{attribute 'Tc2GvlVarNames'}
{attribute 'strict'}
//Stato del WorkAreaManager
TYPE e_Stato_WorkArea :
(
	WORKAREA_STATE_FREE_ENABLED					:= 0,	//WA senza pallet e Abilitata
	WORKAREA_STATE_FREE_DISABLED				:= 1,	//WA senza pallet e disabilitata
	WORKAREA_STATE_OCCUPIED_DISABLED			:= 2,	//WA con pallet e disabilitata
	WORKAREA_STATE_FREE_WORKING					:= 3,	//WA senza pallet e in lavorazione
	WORKAREA_STATE_OCCUPIED_WORKING				:= 4,	//WA con pallet e in lavorazione	
	WORKAREA_STATE_OCCUPIED_WORKED				:= 5, 	//WA con pallet e pallettizzazione terminata
	WORKAREA_STATE_OCCUPIED_WORKED_DISABLED		:= 6,	//WA con pallet e pallettizzazione terminata e area disabilitata
	WORKAREA_STATE_OCCUPIED_TAPING				:= 7,	//WA con pallet in richiesta di nastratura
	WORKAREA_STATE_OCCUPIED_TAPING_DISABLED		:= 8,	//WA con pallet in richiesta di nastratura e area disabilitata
	WORKAREA_STATE_OCCUPIED_TAPED				:= 9,	//WA con pallet e nastratura terminata
	WORKAREA_STATE_OCCUPIED_TAPED_DISABLED		:= 10,	//WA con pallet e nastratura terminata e area disabilitata
	WORKAREA_STATE_OCCUPIED_ENDED				:= 11, 	//WA con pallet e lavorazione terminata
	WORKAREA_STATE_OCCUPIED_ENDED_DISABLED		:= 12, 	//WA con pallet e lavorazione terminata e area disabilitata
	WORKAREA_STATE_OCCUPIED_LGVREQ				:= 13, 	//WA con pallet e richiesta TGV in ingresso
	WORKAREA_STATE_OCCUPIED_LGVREQ_DISABLED		:= 14, 	//WA con pallet e richiesta TGV in ingresso e area disabilitata
	WORKAREA_STATE_OCCUPIED_LGVIN				:= 15, 	//WA con pallet e TGV in ingombro
	WORKAREA_STATE_OCCUPIED_LGVIN_DISABLED		:= 16, 	//WA con pallet e TGV in ingombro e area disabilitata
	WORKAREA_STATE_OCCUPIED_LGVEND				:= 17, 	//WA con pallet e TGV fuori ingombro e Pallet estratto
	WORKAREA_STATE_OCCUPIED_LGVEND_DISABLED		:= 18, 	//WA con pallet e TGV fuori ingombro e Pallet estratto e area disabilata
	WORKAREA_STATE_OCCUPIED_LGVREQ_ABORT        := 19, 	//WA con pallet e richiesta TGV ABORTITA
	
	WORKAREA_STATE_FREE_LGVREQ					:= 20, 	//WA SENZA SUPPORTO e richiesta TGV in ingresso
	WORKAREA_STATE_FREE_LGVREQ_DISABLED			:= 21, 	//WA SENZA SUPPORTO e richiesta TGV in ingresso e area disabilitata
	WORKAREA_STATE_FREE_LGVIN					:= 22, 	//WA SENZA SUPPORTO e TGV in ingombro
	WORKAREA_STATE_FREE_LGVIN_DISABLED			:= 23, 	//WA SENZA SUPPORTO e TGV in ingombro e area disabilitata
	WORKAREA_STATE_FREE_LGVEND					:= 24, 	//WA SENZA SUPPORTO e TGV fuori ingombro e Pallet estratto
	WORKAREA_STATE_FREE_LGVEND_DISABLED			:= 25, 	//WA SENZA SUPPORTO e TGV fuori ingombro e Pallet estratto e area disabilata
	WORKAREA_STATE_FREE_LGVREQ_ABORT        	:= 26, 	//WA SENZA SUPPORTO e richiesta TGV ABORTITA
	
	WORKAREA_STATE_ERROR						:= 99	//WA in errore
);
END_TYPE

(* stored: Version 1.1.0.1, ProductVersion 3.1.4024.11
   EnumerationTextList e_Stato_WorkArea: Id {99cd3464-07f6-477e-9c3c-c778b9481b1d} *)
